{attribute 'qualified_only'}
{attribute 'strict'}
TYPE E_STATES :
(
	Starting := 0,
	Started,
	Stopping,
	Stopped
	
);
END_TYPE

(* stored: Version 1.1.0.1, ProductVersion 3.1.4024.3
   DUT E_STATES: Id {916cea4a-351b-4de0-8d28-48f5d1a03bd7} *)
